(* Logix 5000 project; controller Convert Emulate 5570 rev 36.11; software revision 36.00 *)

TASK MainTask (continuous, watchdog 500 ms) : MainProgram

MODULES
   Local : Emulate 5570 (ICP 2, rev 36.11)
       : 1756-IB16 (ICP 3, rev 3.1, Input RPI 20 ms)
       : 1756-IB16 (ICP 5, rev 3.1, Input RPI 20 ms)
       : vendor 1 type 7 code 16 (ICP 4, rev 3.1, Output RPI 20 ms)
END_MODULES

VAR_GLOBAL   (* controller tags *)
   CONVERT_PB : ALIAS FOR Local:3:I.Data.14;   // Convert Temperature N.O. pushbutton
   ERROR_DUP_VAL : ALIAS FOR Local:4:O.Data.0;   // Error Indicator
   ERROR_OVER_VAL : ALIAS FOR Local:4:O.Data.1;   // Data Error, Over Value
   H_INDC : ALIAS FOR Local:4:O.Data.5;   // High Indicator
   HH_INDC : ALIAS FOR Local:4:O.Data.6;   // High High Indicator
   L_INDC : ALIAS FOR Local:4:O.Data.3;   // Low Indicator
   LL_INDC : ALIAS FOR Local:4:O.Data.2;   // Low Low Indicator
   M_INDC : ALIAS FOR Local:4:O.Data.4;   // Mid Indicator
   RESET_PB : ALIAS FOR Local:3:I.Data.15;   // Data Error Reset, N.O. pushbutton
   TWS_INPUT : ALIAS FOR Local:5:I.Data;   // Thumbwheel Switch
END_VAR

PROGRAM MainProgram   (* main routine TextRoutine *)
VAR
   C_TEMP : DINT;   // Celsius Temperature
   C_TEMP_CONVERT : DINT;   // Celsius Temperature Parameter
   C_TEMP_STORAGE : DINT;   // Storage of Celsius Temperature
   F_TEMP : DINT;   // Fahrenheit Value
   F_TEMP_CONVERT : DINT;   // Fahrenheit Temperature Parameter
   HMI_CONVERT_PB : BOOL;   // HIM CONVERT BUTTON
   HMI_ENABLE_DISABLE : BOOL;   // HMI Enable/Disable Button
   HMI_RESET_PB : BOOL;   // HMI RESET BUTTON
   ONE_SHOT_CONTROL : FBD_ONESHOT;   // One Shot
END_VAR

ROUTINE ConvertBCDRoutine   (* ladder *)
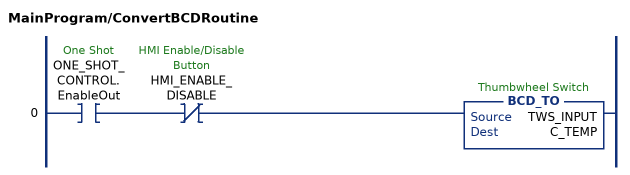
   0: XIC(ONE_SHOT_CONTROL.EnableOut)XIO(HMI_ENABLE_DISABLE)BCD_TO(TWS_INPUT,C_TEMP);
END_ROUTINE

ROUTINE ConvertRoutine   (* structured text *)
   //Convert a Celsius temperature to a Fahrenheit temperature.
   
   //Input Parameter
   SBR(C_TEMP_CONVERT);
   
   F_TEMP_CONVERT := (C_TEMP_CONVERT * 9)/ 5 + 32;
   
   //Return Parameter
   RET(F_TEMP_CONVERT);
END_ROUTINE

ROUTINE IndicatorsRoutine   (* structured text *)
   //Select Case to set range indicator.
   Case F_TEMP of
   	32..49:   LL_INDC := 1;
   		      L_INDC := 0;
   			  M_INDC := 0;
   			  H_INDC := 0;
   			  HH_INDC := 0;
   
   	50..99:   LL_INDC := 0;
   		      L_INDC := 1;
   			  M_INDC := 0;
   			  H_INDC := 0;
   			  HH_INDC := 0;
   
   	100..149:  LL_INDC := 0;
   		      L_INDC := 0;
   			  M_INDC := 1;
   			  H_INDC := 0;
   			  HH_INDC := 0;
   
   	150..199:  LL_INDC := 0;
   		      L_INDC := 0;
   			  M_INDC := 0;
   			  H_INDC := 1;
   			  HH_INDC := 0;
   
   
   	 200..212:  LL_INDC := 0;
   		      L_INDC := 0;
   			  M_INDC := 0;
   			  H_INDC := 0;
   			  HH_INDC := 1;
   
   
   end_case;
END_ROUTINE

ROUTINE InputControlRoutine   (* structured text *)
   //One shot for CONVERT PUSHBUTTON or HMI CONVERT PUSHBUTTON.
   ONE_SHOT_CONTROL.InputBit := HMI_CONVERT_PB OR CONVERT_PB ;
   OSRI(ONE_SHOT_CONTROL);
   
   //Subroutine call if Thumb Wheel Switches are enabled.
   If NOT HMI_ENABLE_DISABLE & ONE_SHOT_CONTROL.OutputBit then
   JSR(ConvertBCDRoutine);
   end_if;
   
   /*If no previous Errors, check for Duplicate or Over Values  and set alarms.*/
   If ONE_SHOT_CONTROL.OutputBit & NOT ERROR_DUP_VAL & NOT ERROR_OVER_VAL then
   	//Check last and current
   	ERROR_DUP_VAL := C_TEMP = C_TEMP_STORAGE;
   	//Check over value
   	ERROR_OVER_VAL := C_TEMP > 100;
   end_if;
   
   
   //Error RESET PUSHBUTTON or HMI RESET PUSHBUTTON and clearing alarms.
   If RESET_PB OR HMI_RESET_PB then
   	ERROR_DUP_VAL := 0;
   	ERROR_OVER_VAL := 0;
   end_if;
   
   /* If no errors, store the celsius value and call the conversion
   routine with the CElsius temperature to return the Fahrenheit
   temperature. */
   If ONE_SHOT_CONTROL.OutputBit & NOT ERROR_DUP_VAL & NOT ERROR_OVER_VAL then
   	C_TEMP_STORAGE := C_TEMP;
   	JSR(ConvertRoutine,1,C_TEMP,F_TEMP);
   end_if;
   
END_ROUTINE

ROUTINE TextRoutine   (* structured text *)
   
   //An unconditional Jump to Subroutine to InputControlRoutine.
   //An unconditional Jump to Subroutine to IndicatorsRoutine
   JSR(InputControlRoutine);
   JSR(IndicatorsRoutine);
   
   
END_ROUTINE
END_PROGRAM
